Fanuc KAREL source: IO0098.KL

PROGRAM IO0098
%STACKSIZE=65535
%PRIORITY=65535
%NOLOCKGROUP
ROUTINE RTEST FROM IO0098
ROUTINE RTEST
VAR
L1 : ARRAY[3] OF INTEGER
L2 : XYZWPR
L3 : JOINTPOS9
L4 : POSITION
U2C_37 : BOOLEAN -- ASSUMED 2C source type; see uncertainty report
U2C_38 : REAL -- ASSUMED 2C source type; see uncertainty report
U2C_39 : REAL -- ASSUMED 2C source type; see uncertainty report
U2C_40 : INTEGER -- ASSUMED 2C source type; see uncertainty report
U2C_41 : INTEGER -- ASSUMED 2C source type; see uncertainty report
BEGIN
U2C_37=TRUE
L1[1]=2
U2C_40=1
U2C_41=1065353216
-- UNSAFE_SOURCE_IR line 19: FRAME[RTEST+0x28] = native_io_value(8, 17)
END RTEST
BEGIN
RTEST
END IO0098
